# B&R Automation Studio project betaautomationstudio
Automation Studio 4.9.2.46; technology packages: Acp10Arnc0 5.12.2

## Configuration Config1

CPU X20CP1586, AutomationRuntime C4.90, Build 4.1.2, Vc V4.72.2

### Task classes (Cpu.sw)
```
Cyclic#4:
  control <- control.prg
  varUpdates <- varUpdates.prg
NcDataObjects: acp10etxen <- acp10etxen.dob, gAxisa <- gAxisobj.gAxisa.dob, gAxisi <- gAxisobj.gAxisi.dob
VcDataObjects: Visu <- Visu.dob
Libraries: Acp10man, Acp10par, NcGlobal, Acp10_MC, sys_lib, brsystem, runtime, Acp10sim
```

### Hardware
```
X20CP1586 : X20CP1586 v1.8.1.0
  Connector IF2:
    ActivateDevice = 1
    Vnc1
    VncVcObjectName1 = Visu
    VncKeyMappingFile1 = VC\PS2-Keyboard.dis
  ConfigurationID = betaprojectAS_Config1
  Simulation = 1
```

### Acp10cfg.ncc - X20CP1586/Motion/Acp10cfg.ncc
```
NcConfiguration (Version=5.12.2, NcSwId=Acp10)
  ACP10CF1_typ:
    cnt_nettrc_rec_drive = 1500
    bufsize_trace_upload = 1200
    tc_nc_man_task = Cyclic #1
    glob_pv_as_ncobject = Yes
    ncsys_dl_broadcast = Yes
    ncsys_dl_acp_reset = Yes
    safemc_log_err_to_ax = Yes
    network_init:
      ncsw_init_execute = Yes
      automatic_execute = No
      node_nr_warning = Yes
      net_err_before_ncact = Yes
    nettrc:
      enter_parsecrec = Yes
      enter_ncaction = Yes
      save_ring_startidx = Yes
    cam_prof_download:
      cam_dat_dl_parallel = No
      tc_cam_dl_parallel = Task class for NC Manager task
    plk_if[0]:
      if_name = IF3
      tc_CycDat_PLCopen = Task class for NC Manager task
      mc_broadcast_extdat = No
```

### Acp10map.ncm - X20CP1586/Motion/Acp10map.ncm
```
NcMapping (NcSwId=Acp10, DisabledNodesAreHidden=False)
  NcObject gAxis (ModuleId=8EIxxxMxS1x.xxxx-1, Type=ncAXIS, Channel=1, AcoposSimulation=Standard, InitParameter=gAxisi, AcoposParameter=gAxisa, Disabled=FALSE, ModuleDisabled=FALSE)
  NcObject 8EIxxxMxS1x.xxxx-1_ncV_AXIS1 (ModuleId=8EIxxxMxS1x.xxxx-1, Type=ncV_AXIS, Channel=1, Disabled=TRUE, ModuleDisabled=FALSE)
```

### PvMap.vvm - X20CP1586/PvMap.vvm
```iecst
VAR_CONFIG
	::pvi AT %Q.::pvi; (*PVI Variables, lol*)
END_VAR
```

## Logical view

Binary libraries used (declarations not repeated): operator, runtime, astime, AsIecCon, Acp10man 5.12.2, Acp10par 5.12.2, NcGlobal 5.12.2, Acp10_MC 5.12.2, sys_lib, brsystem, Acp10sim 5.12.2

### Global.typ - Global data types
```iecst
TYPE
	ctrlStateEnum :
		(
		CTRL_INIT,
		CTRL_OFF,
		CTRL_POWER_ON_AXIS,
		CTRL_POWERING_ON_AXIS,
		CTRL_POWER_OFF_AXIS,
		CTRL_POWERING_OFF_AXIS,
		CTRL_HOME_AXIS,
		CTRL_HOMING_AXIS,
		CTRL_STOPPING,
		CTRL_STANDSTILL,
		CTRL_MOVE_VELOCITY,
		CTRL_MOVE_ABSOLUTE,
		CTRL_ERROR,
		CTRL_MOVE_VELOCITY_ERROR,
		CTRL_MOVE_ABSOLUTE_ERROR,
		CTRL_FATAL_ERROR,
		CTRL_FATAL_ERROR_EXIT
	);

	mcBlocksType : STRUCT
		power : MC_Power;
		home : MC_Home;
		stop : MC_Stop;
		reset : MC_Reset;
		moveVelocity : MC_MoveVelocity;
		moveAbsolute : MC_MoveAbsolute;
		currentPosition : MC_ReadActualPosition;
		currentVelocity : MC_ReadActualVelocity;
		status : MC_ReadStatus;
		error : MC_ReadAxisError;
	END_STRUCT;

	gLocalPID : STRUCT
		enabled : BOOL;					(*  *)
		proportionalGain : BOOL;		(*  *)
		integralGain : BOOL;			(*  *)
		derivativeGain : BOOL;			(*  *)
	END_STRUCT;

	gControlType : STRUCT
		localPID : gLocalPID;			(*  *)
		modeVelocity : BOOL;			(*  *)
		setPosition : REAL;				(*  *)
		setDirection : BOOL;			(*  *)
		setVelocity : REAL;				(*  *)
		currentPosition : REAL;			(*  *)
		currentAngle : REAL;			(*  *)
		currentVelocity : REAL;			(*  *)
		currentDirection : INT;			(*  *)
		limitAcceleration : REAL := 1000;	(*  *)
		limitVelocity : REAL := 200;	(*  *)
		limitPosPos : DINT := -5000;	(*  *)
		limitNegPos : DINT := 5000;		(*  *)
	END_STRUCT;

	hmiType : STRUCT
		fields : vFieldType;			(*  *)
		indicators : vIndicatorType;	(*  *)
		buttons : vButtonType;			(*  *)
	END_STRUCT;

	vButtonType : STRUCT
		on : BOOL;						(*  *)
		onPrevious : BOOL;
		off : BOOL;						(*  *)
		offPrevious : BOOL;
		start : BOOL;					(*  *)
		startPrevious : BOOL;
		stop : BOOL;					(*  *)
		stopPrevious : BOOL;
		localPid : BOOL;				(*  *)
		localPidPrevious : BOOL;
		simulinkPid : BOOL;				(*  *)
		simulinkPidPrevious : BOOL;
		externalSim : BOOL;				(*  *)
		externalSimPrevious : BOOL;
		simulinkSim : BOOL;				(*  *)
		simulinkSimPrevious : BOOL;
		ackError : BOOL;				(*  *)
		ackErrorPrevious : BOOL;
		overridePosition : BOOL;		(*  *)
		overridePositionPrevious : BOOL;
	END_STRUCT;

	vFieldType : STRUCT
		velocity : REAL;			(*  *)
		position : REAL;			(*  *)
		angle : REAL;				(*  *)
		ovrPosition : REAL;			(*  *)
		accelerationLimit : REAL;	(*  *)
		velocityLimit : REAL;		(*  *)
		positionLimitNeg : DINT;	(*  *)
		positionLimitPos : DINT;	(*  *)
		controlState : WSTRING[40];	(*  *)
		errorCode : REAL;			(*  *)
		errorText : WSTRING[40];	(*  *)
	END_STRUCT;

	vIndicatorType : STRUCT
		power : INT;				(*  *)
		home : INT;					(*  *)
		stop : INT;					(*  *)
		reset : INT;				(*  *)
		moveVelocity : INT;			(*  *)
		movePosition : INT;			(*  *)
		readVelocity : INT;			(*  *)
		readPosition : INT;			(*  *)
		status : INT;				(*  *)
		error : INT;				(*  *)
		readParam : INT;			(*  *)
		writeParam : INT;			(*  *)
	END_STRUCT;

	opcuaWriteType : STRUCT 			(* For variables read from OPCUA *)
		cartPosition : REAL := 0.0;		(* mm *)
		cartVelocity : REAL := 0.0;		(* mm/s *)
		pendulumAngle : REAL := 0.0;	(* Rad, 0 is upright position *)
	END_STRUCT;
	opcuaReadType : STRUCT 				(* For variables written to OPCUA *)
		setCartVelocity : REAL := 0.0;	(* Negative is backward motion *)
	END_STRUCT;

	pviMotorType : STRUCT
		start : BOOL := FALSE;				(* Start the motor *)
		forward : BOOL := FALSE;			(* Set motor direction *)
		setVelocity : INT := 0;				(*  *)
		setConverterFrequency : INT := 0;	(*  *)
		isStarted : BOOL := FALSE;			(*  *)
		isStopped : BOOL := FALSE;			(*  *)
		isForward : BOOL := FALSE;			(*  *)
		isBackward : BOOL := FALSE;			(*  *)
		isMax : BOOL := FALSE;				(* Motor is at max limit *)
		isMiddle : BOOL := FALSE;			(* Motor is on exact middle *)
		isMin : BOOL := FALSE;				(* Motor is at min limit *)
		offsetMax : BOOL := FALSE;			(*  *)
		offsetMin : BOOL := FALSE;			(*  *)
		isReset : BOOL := FALSE;			(*  *)
		velocity : INT := 0;				(* Actual motor velocity *)
	END_STRUCT;

	pviType : STRUCT
		cartPositionEncoder : DINT := 0;	(* Cart position encoder output, currently in 1mm/units *)
		pendulumAngle : DINT := 0; 		(* Angle output, 1024 divisions per rotation *)
		motor : pviMotorType;		(* All motor specific variables *)
	END_STRUCT;

END_TYPE
```

### Global.var - Global variables
```iecst
VAR
	gAxis : ACP10AXIS_typ;			(* Required axis object *)

	ctrlState : ctrlStateEnum := CTRL_INIT;	(* Control loop state *)
	mc : mcBlocksType;				(* Function blocks for motor control *)

	gControl : gControlType;		(* Control related variables *)
	hmi : hmiType;					(* HMI stuff *)
	opcua_r : opcuaReadType;		(* Variables readable with OPCUA *)
	opcua_w : opcuaWriteType;		(* Variables writeable with OPCUA *)
	pvi : pviType;					(* Variables shared with PVI *)
END_VAR
```


### Data object Logical/acp10etxen (Ett)

- acp10etxen.ett (not shown)

### Package Logical/gAxisobj - gAxisobj

- Data object Logical/gAxisobj/gAxisa (Apt) (no source held here)

### Data object Logical/gAxisobj/gAxisi (Ax)

#### gAxisi.ax
```
InitParameter (Version=5.12.2, NcSwId=Acp10)
  ACP10AXIS_typ:
    dig_in:
      level:
        reference = ncACTIV_HI
        pos_hw_end = ncACTIV_HI
        neg_hw_end = ncACTIV_HI
        trigger1 = ncACTIV_HI
        trigger2 = ncACTIV_HI
    encoder_if:
      parameter:
        count_dir = ncSTANDARD
        scaling:
          load:
            units = 1000
            rev_motor = 1
    limit:
      parameter:
        v_pos = 10000
        v_neg = 10000
        a1_pos = 50000
        a2_pos = 50000
        a1_neg = 50000
        a2_neg = 50000
        t_jolt = 0
        t_in_pos = 0
        pos_sw_end = 2000000000
        neg_sw_end = -2000000000
        ds_warning = 500
        ds_stop = 1000
        a_stop = 1.0e30
        dv_stop = 0
        dv_stop_mode = ncOFF
    controller:
      mode = ncPOSITION
      position:
        kv = 50
        tn = 0
        t_predict = 0.0004
        t_total = 0.0004
        p_max = 1.0e30
        i_max = 0
      speed:
        kv = 2.0
        tn = 0
        t_filter = 0.0
        isq_filter1:
          type = ncOFF
          a0 = 0.0
          a1 = 0.0
          b0 = 0.0
          b1 = 0.0
          b2 = 0.0
          c0_par_id = 0
          c1_par_id = 0
        isq_filter2:
          type = ncOFF
          a0 = 0.0
          a1 = 0.0
          b0 = 0.0
          b1 = 0.0
          b2 = 0.0
          c0_par_id = 0
          c1_par_id = 0
        isq_filter3:
          type = ncOFF
          a0 = 0.0
          a1 = 0.0
          b0 = 0.0
          b1 = 0.0
          b2 = 0.0
          c0_par_id = 0
          c1_par_id = 0
      uf:
        type = ncLINEAR + ncCORRECTION
        auto_config = ncMOTOR_PAR
        u0 = 0
        un = 0
        fn = 50.0
        k_f_slip = 0
      ff:
        mode = ncSTANDARD
        torque_load = 0.0
        torque_pos = 0.0
        torque_neg = 0.0
        kv_torque = 0.0
        inertia = 0.0
        t_filter_a = 0.0
      fb:
        mode = ncSTANDARD
        speed_mix_ratio = 0.0
        speed_kv = 2.0
      model:
        mass1:
          inertia = 0
          viscous_friction = 0
        mass2:
          inertia = 0
          viscous_friction = 0
          stiffness = 0
          damping = 0
    move:
      stop:
        parameter[0]:
          decel_ramp = ncA_LIMIT
          controller = ncON
        parameter[1]:
          decel_ramp = ncA_LIMIT
          controller = ncON
        parameter[2]:
          decel_ramp = ncA_LIMIT
          controller = ncON
        parameter[3]:
          decel_ramp = ncA_LIMIT
          controller = ncON
        quickstop:
          decel_ramp = ncA_LIMIT
          t_jolt = 0
        drive_error:
          decel_ramp = ncA_LIMIT
      homing:
        parameter:
          s = 0
          v_switch = 5000
          v_trigger = 500
          a = 50000
          mode = ncDIRECT
          edge_sw = ncPOSITIVE
          start_dir = ncPOSITIVE
          trigg_dir = ncPOSITIVE
          ref_pulse = ncOFF
          fix_dir = ncOFF
          tr_s_block = 0
          torque_lim = 0
          ds_block = 0
          ds_stop = 0
      basis:
        parameter:
          v_pos = 5000
          v_neg = 5000
          a1_pos = 50000
          a2_pos = 50000
          a1_neg = 50000
          a2_neg = 50000
    message:
      text:
        parameter:
          format = ncBREAK
          columns = 80
          data_modul = acp10etxen
```

### Program Logical/control (IEC)

#### Variables.var
```iecst
VAR
	state : ctrlStateEnum := CTRL_INIT;
	mc : mcBlocksType;
END_VAR
```

#### Main.st
```iecst
PROGRAM _INIT
	(* Insert code here *)

END_PROGRAM

PROGRAM _CYCLIC
	CASE ctrlState OF
		CTRL_INIT:
			// Binding the motion axis to MC blocks
			mc.home.Axis := ADR(gAxis);
			mc.moveAbsolute.Axis := ADR(gAxis);
			mc.moveVelocity.Axis := ADR(gAxis);
			mc.power.Axis := ADR(gAxis);
			mc.reset.Axis := ADR(gAxis);
			mc.stop.Axis := ADR(gAxis);
			mc.currentPosition.Axis := ADR(gAxis);
			mc.currentVelocity.Axis := ADR(gAxis);
			mc.error.Axis := ADR(gAxis);

			// Next state
			ctrlState := CTRL_OFF;

		CTRL_OFF:
			// Check if ON is requested and change state
			IF hmi.buttons.on THEN
				ctrlState := CTRL_POWER_ON_AXIS;
			END_IF

		CTRL_POWER_ON_AXIS:
			// Enable the block required for std operation
			mc.power.Enable := TRUE;
			mc.currentPosition.Enable := TRUE;
			mc.currentVelocity.Enable := TRUE;
			mc.error.Enable := TRUE;
			mc.status.Enable := TRUE;

			// Change state
			ctrlState := CTRL_POWERING_ON_AXIS;

		CTRL_POWERING_ON_AXIS:
			// Change state if Power is on
			// TODO: Include checks for the other blocks?
			IF mc.power.Status THEN
				ctrlState := CTRL_HOME_AXIS;
			END_IF

		CTRL_POWER_OFF_AXIS:
			// Disable the blocks used for std operation
			mc.power.Enable := FALSE;
			mc.currentPosition.Enable := FALSE;
			mc.currentVelocity.Enable := FALSE;
			mc.error.Enable := FALSE;
			mc.status.Enable := FALSE;

			// Change state
			ctrlState := CTRL_POWERING_OFF_AXIS;

		CTRL_POWERING_OFF_AXIS:
			// Change state when block are off
			IF NOT mc.power.Status AND NOT mc.currentPosition.Valid AND NOT mc.currentVelocity.Valid THEN
				ctrlState := CTRL_OFF;
			END_IF

		CTRL_HOME_AXIS:
			// If Execute is true, flip and come back next cycle
			IF mc.home.Execute THEN
				mc.home.Execute := FALSE;
			ELSE
				// Start homing and change state
				mc.home.Execute := TRUE;
				ctrlState := CTRL_HOMING_AXIS;
			END_IF

		CTRL_HOMING_AXIS:
			// Change state when homing is done
			IF mc.home.Done THEN
				mc.home.Execute := FALSE;
				ctrlState := CTRL_STOPPING;
			END_IF

		CTRL_STOPPING:
			// Change state when confirmed stopped
			mc.stop.Execute := TRUE;
			IF mc.stop.Done THEN
				mc.stop.Execute := FALSE;
				ctrlState := CTRL_STANDSTILL;
			END_IF

		CTRL_STANDSTILL:
			// Wait for something to start the operation
			IF hmi.buttons.start OR hmi.buttons.overridePosition THEN
				// Reset the button
				hmi.buttons.start := FALSE;
				// If the override move position is active, do that
				IF hmi.buttons.overridePosition THEN
					// Set the move position from the field
					gControl.setPosition := hmi.fields.ovrPosition;
					// Reset the button
					hmi.buttons.overridePosition := FALSE;
					// Change to move absolute state
					ctrlState := CTRL_MOVE_ABSOLUTE;
				ELSE
					// 'Normal' velocity based operation
					ctrlState := CTRL_MOVE_VELOCITY;
				END_IF
			ELSIF hmi.buttons.off THEN
				// Power off if button has been pushed
				hmi.buttons.off := FALSE;
				ctrlState := CTRL_POWER_OFF_AXIS;
			END_IF

		CTRL_MOVE_VELOCITY:
			// Check if a stop or manual position override is requested
			IF hmi.buttons.stop OR hmi.buttons.overridePosition THEN
				// Reset button
				hmi.buttons.stop := FALSE;
				// Stop velocity block and change to stop state
				mc.moveVelocity.Execute := FALSE;
				ctrlState := CTRL_STOPPING;
			ELSE
				// Check that velocity requested is within limits
				IF gControl.setVelocity >= 0 AND gControl.setVelocity < gControl.limitVelocity THEN
					// Update move block velocity
					mc.moveVelocity.Velocity := gControl.setVelocity;
					// Set direction
					IF gControl.setDirection THEN
						mc.moveVelocity.Direction := mcPOSITIVE_DIR;
					ELSE
						mc.moveVelocity.Direction := mcNEGATIVE_DIR;
					END_IF

					// Toggle execute and update the block to allow for changes in same cycle
					IF mc.moveVelocity.Execute THEN
						mc.moveVelocity.Execute := FALSE;
						mc.moveVelocity();
					END_IF
					// Start executing move
					mc.moveVelocity.Execute := TRUE;
				ELSE
					// Limits not met, stop motion
					mc.moveVelocity.Velocity := 0;
					mc.moveVelocity.Execute := FALSE;
					ctrlState := CTRL_STOPPING;
				END_IF
			END_IF

		CTRL_MOVE_ABSOLUTE:
			// This move mode is used for the override position only
			IF hmi.buttons.stop THEN
				// Reset the button
				hmi.buttons.stop := FALSE;
				// Stop moving
				mc.moveAbsolute.Execute := FALSE;
				ctrlState := CTRL_STOPPING;
			ELSIF mc.moveAbsolute.Done THEN
				// Movement complete, go to standstill state
				mc.moveAbsolute.Execute := FALSE;
				ctrlState := CTRL_STANDSTILL;
			ELSE
				// Check if move is needed (within 0.1 unit of current position)
				IF ABS(gControl.currentPosition - gControl.setPosition) > 0.1 THEN
					// Set new position in block
					mc.moveAbsolute.Position := gControl.setPosition;
					// Start execution
					mc.moveAbsolute.Execute := TRUE;
				ELSIF NOT mc.moveAbsolute.Execute THEN
					// Move not big enough, go to standstill state
					// If block is already active we might just be very close and don't want to do anything
					mc.moveAbsolute.Execute := FALSE;
					ctrlState := CTRL_STANDSTILL;
				END_IF
			END_IF

		CTRL_ERROR:

		CTRL_FATAL_ERROR:

		CTRL_FATAL_ERROR_EXIT:

	END_CASE

	// Updating blocks, minus info-only blocks (see varUpdates loop)
	mc.home();
	mc.moveAbsolute();
	mc.moveVelocity();
	mc.power();
	mc.reset();
	mc.stop();

	// Error checking
	// TODO: Do something
	IF mc.home.Error THEN
	END_IF
	IF mc.moveAbsolute.Error THEN
	END_IF
	IF mc.moveVelocity.Error THEN
	END_IF
	IF mc.power.Error THEN
	END_IF
	IF mc.reset.Error THEN
	END_IF
	IF mc.stop.Error THEN
	END_IF
	IF mc.currentPosition.Error THEN
	END_IF
	IF mc.currentVelocity.Error THEN
	END_IF
	IF mc.status.Error THEN
	END_IF

END_PROGRAM

PROGRAM _EXIT
	(* Insert code here *)

END_PROGRAM
```

- Visualisation Logical/Visu (not shown)

### Program Logical/varUpdates (IEC)

#### Main.st
```iecst
PROGRAM _INIT
	(* Insert code here *)

END_PROGRAM

PROGRAM _CYCLIC
	// Clearing errorText if ack'ed
	IF hmi.buttons.ackError THEN
		// Reset button
		hmi.buttons.ackError := FALSE;
		// Acknowledge error
		mc.error.Acknowledge := TRUE;
	END_IF

	// Update the function blocks used for errors and reading values
	mc.currentPosition();
	mc.currentVelocity();
	mc.status();
	mc.error();

	// Some HMI button logic for determining which sim and PID to use
	IF hmi.buttons.externalSim AND NOT hmi.buttons.externalSimPrevious THEN
		// Mode switched to external sim
		hmi.buttons.externalSimPrevious := hmi.buttons.externalSim;
		hmi.buttons.simulinkSim := NOT hmi.buttons.externalSim;
		hmi.buttons.simulinkSimPrevious := NOT hmi.buttons.externalSim;
	END_IF
	IF hmi.buttons.simulinkSim AND NOT hmi.buttons.simulinkSimPrevious THEN
		// Mode switched to simulink sim
		hmi.buttons.simulinkSimPrevious := hmi.buttons.simulinkSim;
		hmi.buttons.externalSim := NOT hmi.buttons.simulinkSim;
		hmi.buttons.externalSimPrevious := NOT hmi.buttons.simulinkSim;
	END_IF

	IF hmi.buttons.localPid AND NOT hmi.buttons.localPidPrevious THEN
		// Mode switched to local PID
		hmi.buttons.localPidPrevious := hmi.buttons.localPid;
		hmi.buttons.simulinkPid := NOT hmi.buttons.localPid;
		hmi.buttons.simulinkPidPrevious := NOT hmi.buttons.localPid;
	END_IF
	IF hmi.buttons.simulinkPid AND NOT hmi.buttons.simulinkPidPrevious THEN
		// Mode switched to simulink PID
		hmi.buttons.simulinkPidPrevious := hmi.buttons.simulinkPid;
		hmi.buttons.localPid := NOT hmi.buttons.simulinkPid;
		hmi.buttons.localPidPrevious := NOT hmi.buttons.simulinkPid;
	END_IF

	// Update variables from motor position, velocity, and pendulum angle
	gControl.currentAngle := 0; // TODO: Where do I get this?
	gControl.currentPosition := mc.currentPosition.Position;
	gControl.currentVelocity := mc.currentVelocity.Velocity;
	gControl.currentDirection := mc.moveVelocity.Direction;

	// Update variables from simulation through PVI
	IF hmi.buttons.externalSim THEN
		// Read the current pendulum angle and cart position? from PVI
		// TODO: Scale this correctly
		gControl.currentAngle := DINT_TO_REAL(pvi.pendulumAngle);
		// TODO: I don't think we should let pvi override the MC block position?
		//gControl.currentPosition := pvi.cartPositionEncoder;
		// Write the current motor state, direction and velocity to PVI
		pvi.motor.start := mc.moveVelocity.Execute;
		pvi.motor.setVelocity := REAL_TO_INT(mc.moveVelocity.Velocity);
		IF mc.moveVelocity.Direction = mcPOSITIVE_DIR THEN
			pvi.motor.forward := TRUE;
		ELSE
			pvi.motor.forward := FALSE;
		END_IF

	END_IF
	// Update variables for simulink simulation
	IF hmi.buttons.simulinkSim THEN
		// Read the current pendulum angle from OPCUA
		gControl.currentAngle := opcua_w.pendulumAngle;
		// Write the position and cart velocity to OPCUA
		// TODO: Scale the written velocity correctly
		opcua_w.cartPosition := gControl.currentPosition;
		opcua_w.cartVelocity := gControl.currentVelocity;
	END_IF

	// Update variables for local PID control?
	IF hmi.buttons.localPid THEN
	END_IF
	// Update variables for simulink PID control
	IF hmi.buttons.simulinkPid THEN
		// Write the current position and angle
		// Read the new setVelocity
		gControl.setVelocity := opcua_r.setCartVelocity;
		// Write the current position and pendulum angle to OPCUA
		opcua_w.cartPosition := gControl.currentPosition;
		// TODO: Map the velocity correctly
		opcua_w.cartVelocity := gControl.currentVelocity;
		opcua_w.pendulumAngle := gControl.currentAngle;
	END_IF

	// Set movement limits from gControl struct
	mc.moveAbsolute.Acceleration := gControl.limitAcceleration;
	mc.moveAbsolute.Deceleration := gControl.limitAcceleration;
	mc.moveAbsolute.Velocity := gControl.limitVelocity;
	mc.moveVelocity.Acceleration := gControl.limitAcceleration;
	mc.moveVelocity.Deceleration := gControl.limitAcceleration;

	// And an error block thing
	mc.error.Acknowledge := FALSE;

	// Update HMI fields and indicators
	CASE ctrlState OF
		CTRL_INIT:
			hmi.fields.controlState := "CTRL_INIT";
		CTRL_OFF:
			hmi.fields.controlState := "CTRL_OFF";
		CTRL_POWER_ON_AXIS:
			hmi.fields.controlState := "CTRL_POWER_ON_AXIS";
		CTRL_POWERING_ON_AXIS:
			hmi.fields.controlState := "CTRL_POWERING_ON_AXIS";
		CTRL_POWER_OFF_AXIS:
			hmi.fields.controlState := "CTRL_POWER_OFF_AXIS";
		CTRL_POWERING_OFF_AXIS:
			hmi.fields.controlState := "CTRL_POWERING_OFF_AXIS";
		CTRL_HOME_AXIS:
			hmi.fields.controlState := "CTRL_HOME_AXIS";
		CTRL_HOMING_AXIS:
			hmi.fields.controlState := "CTRL_HOMING_AXIS";
		CTRL_STOPPING:
			hmi.fields.controlState := "CTRL_STOPPING";
		CTRL_STANDSTILL:
			hmi.fields.controlState := "CTRL_STANDSTILL";
		CTRL_MOVE_VELOCITY:
			hmi.fields.controlState := "CTRL_MOVE_VELOCITY";
		CTRL_MOVE_ABSOLUTE:
			hmi.fields.controlState := "CTRL_MOVE_ABSOLUTE";
		CTRL_ERROR:
			hmi.fields.controlState := "CTRL_ERROR";
		CTRL_FATAL_ERROR:
			hmi.fields.controlState := "CTRL_FATAL_ERROR";
		CTRL_FATAL_ERROR_EXIT:
			hmi.fields.controlState := "CTRL_FATAL_ERROR_EXIT";
		ELSE
			hmi.fields.controlState := "State fell through HMI Case!";
	END_CASE

	hmi.fields.errorCode := mc.error.ErrorID;
	hmi.fields.errorText := STRING_TO_WSTRING(mc.error.DataObjectName);

	hmi.fields.accelerationLimit := gControl.limitAcceleration;
	hmi.fields.velocityLimit := gControl.limitVelocity;
	hmi.fields.positionLimitPos := gControl.limitNegPos;
	hmi.fields.positionLimitNeg := gControl.limitPosPos;

	hmi.fields.angle := gControl.currentAngle;
	hmi.fields.position := gControl.currentPosition;
	hmi.fields.velocity := gControl.currentVelocity;

	hmi.indicators.power := mc.power.Error OR NOT mc.power.Enable;
	hmi.indicators.home := mc.home.Error OR NOT mc.home.Busy;
	hmi.indicators.stop := mc.stop.Error OR NOT mc.stop.Busy;
	hmi.indicators.reset := mc.reset.Error OR NOT mc.reset.Execute;
	hmi.indicators.moveVelocity := mc.moveVelocity.Error OR NOT mc.moveVelocity.Execute;
	hmi.indicators.movePosition := mc.moveAbsolute.Error OR NOT mc.moveAbsolute.Execute;
	hmi.indicators.readVelocity := mc.currentVelocity.Error OR NOT mc.currentVelocity.Enable;
	hmi.indicators.readPosition := mc.currentPosition.Error OR NOT mc.currentPosition.Enable;
	hmi.indicators.status := mc.status.Error AND NOT mc.status.Enable;
	hmi.indicators.error := mc.error.Error AND NOT mc.error.Enable;

END_PROGRAM

PROGRAM _EXIT
	(* Insert code here *)

END_PROGRAM
```

### Program Logical/Program

#### Types.typ
```iecst
TYPE
	controlStateEnum : (
		CTRL_INIT,
		CTRL_HOME_START,
		CTRL_HOME_SEEK_NEG,
		CTRL_HOME_SEEK_POS,
		CTRL_HOME_CENTER,
		CTRL_STOP,
		CTRL_RUNNING,
		CTRL_NO_SIM,
		CTRL_NO_CONTROLLER
	);

	opcuaType : STRUCT 			(* For OPCUA *)
		cartPosition : REAL := 0.0;		(* mm *)
		cartVelocity : REAL := 0.0;		(* mm/s *)
		pendulumAngle : REAL := 0.0;	(* Rad, 0 is upright position *)
		setCartVelocity : REAL := 0.0;	(* Negative is backward motion *)
	END_STRUCT;

	pviMotorType : STRUCT
		start : BOOL := FALSE;				(* Start the motor *)
		forward : BOOL := FALSE;			(* Set motor direction *)
		setVelocity : INT := 0;				(*  *)
		setConverterFrequency : INT := 0;	(*  *)
		isStarted : BOOL := FALSE;			(*  *)
		isStopped : BOOL := FALSE;			(*  *)
		isForward : BOOL := FALSE;			(*  *)
		isBackward : BOOL := FALSE;			(*  *)
		isMax : BOOL := FALSE;				(* Motor is at max limit *)
		isMiddle : BOOL := FALSE;			(* Motor is on exact middle *)
		isMin : BOOL := FALSE;				(* Motor is at min limit *)
		offsetMax : BOOL := FALSE;			(*  *)
		offsetMin : BOOL := FALSE;			(*  *)
		isReset : BOOL := FALSE;			(*  *)
		velocity : INT := 0;				(* Actual motor velocity *)
	END_STRUCT;

	pviType : STRUCT
		cartPositionEncoder : DINT := 0;	(* Cart position encoder output, currently in 1mm/units *)
		pendulumAngle : DINT := 0; 		(* Angle output, 1024 divisions per rotation *)
		motor : pviMotorType;			(* All motor specific variables *)
	END_STRUCT;

	controlType : STRUCT
		state : controlStateEnum;		(*  *)
		setVelocity : REAL;				(*  *)
		setPosition : REAL := 0;
		setPointPosition : REAL := 0;
		setAngle : REAL := 0;
		currentPosition : REAL;			(*  *)
		currentAngle : REAL;			(*  *)
		currentVelocity : REAL;			(*  *)
		currentAngularVelocity : REAL;
		currentDirection : BOOL;		(*  *)
		limitAcceleration : REAL := 1000;	(*  *)
		limitVelocity : REAL := 20000;	(*  *)
		limitPosPos : DINT := -5000;	(*  *)
		limitNegPos : DINT := 5000;		(*  *)
		homing : homingType;		(*  *)
	END_STRUCT;

	localLqrType : STRUCT
		A : ARRAY[1..4, 1..4] OF LREAL :=
		0, 1, 0, 0,
		0, -10, 1.6498, -0.0134,
		0, 0, 0, 1,
		0, -55.8140, 64.0173, -0.5198;
		B : ARRAY[1..4] OF LREAL := 0, 2, 0, 11.1628;
		Kf : ARRAY[1..4, 1..2] OF LREAL :=
		-3.1768, -0.0803,
		-0.0491, -1.2372,
		-0.0803, -15.3344,
		-0.2485, -112.5752;
		Klqr2 : ARRAY[1..4] OF LREAL := -3.3541, -12.8984, 57.1684, 16.7280;

		Klqr : ARRAY[1..4] OF LREAL := 2.5683, 9.3490, -38.5829, -12.4979;

		u : LREAL := 0;

		x : ARRAY[1..4] OF LREAL := 0,0,0,0;
		xn : ARRAY[1..4] OF LREAL := 0,0,0,0;

		intOut : ARRAY[1..4] OF LREAL := 0,0,0,0;
		intSave : ARRAY[1..4] OF LREAL := 0,0,0,0;

		mc : LREAL := 0.5;
		mp : LREAL := 0.084;
		Ts : LREAL := 0.01;
	END_STRUCT;

	homingType : STRUCT
		foundNegLim : REAL;				(*  *)
		foundPosLim : REAL;				(*  *)
		seekVelocity : REAL := 500;		(*  *)
		middleVelocity : REAL := 1500;	(*  *)
	END_STRUCT;

	hmiType : STRUCT
		fields : hmiFieldType;			(*  *)
		indicators : hmiIndicatorType;	(*  *)
		buttons : hmiButtonType;			(*  *)

	END_STRUCT;

	hmiButtonType : STRUCT
		start : BOOL;					(*  *)
		startPrevious : BOOL;
		localPid : BOOL;				(*  *)
		localPidPrevious : BOOL;
		simulinkPid : BOOL;				(*  *)
		simulinkPidPrevious : BOOL;
		experiorSim : BOOL;				(*  *)
		experiorSimPrevious : BOOL;
		simulinkSim : BOOL;				(*  *)
		simulinkSimPrevious : BOOL;
	END_STRUCT;

	hmiFieldType : STRUCT
		velocity : REAL;			(*  *)
		position : REAL;			(*  *)
		angle : REAL;				(*  *)
		ovrPosition : REAL;			(*  *)
		accelerationLimit : REAL;		(*  *)
		velocityLimit : REAL;			(*  *)
		positionLimitNeg : REAL;		(*  *)
		positionLimitPos : REAL;		(*  *)
		controlState : WSTRING[40];		(*  *)
	END_STRUCT;

	hmiIndicatorType : STRUCT
		pvi : BOOL; 	(*  *)
		opcua : BOOL;	(*  *)
	END_STRUCT;

END_TYPE
```

#### Variables.var
```iecst
VAR
	control : controlType;
	hmi : hmiType;
	opcua : opcuaType;
	pvi : pviType;
	lqr : localLqrType;
END_VAR
```

#### Main.st
```iecst
PROGRAM _INIT

	// Start in local mode with experior sim
	hmi.buttons.start := TRUE;
	hmi.buttons.experiorSim := TRUE;
	hmi.buttons.localPid := TRUE;

END_PROGRAM

PROGRAM _CYCLIC
	// 1. BUTTON LOGIC
	// 2. SIMULATION READS
	// 3. STATE SWITCH
	// 	3.1 HOMING
	//	3.2 SEEK TO MID
	//	3.3 CONTROL LOOP MODE
	// 4. SIMULATION WRITES
	// 5. HMI

	//////////////////
	// BUTTON LOGIC //
	//////////////////
	// Experior simulation button
	IF hmi.buttons.experiorSim AND NOT hmi.buttons.experiorSimPrevious THEN
		// Mode switched to experior sim
		hmi.buttons.experiorSimPrevious := hmi.buttons.experiorSim;
		hmi.buttons.simulinkSim := NOT hmi.buttons.experiorSim;
		hmi.buttons.simulinkSimPrevious := NOT hmi.buttons.experiorSim;
	ELSIF NOT hmi.buttons.experiorSim AND hmi.buttons.experiorSimPrevious THEN
		// Switched off
		hmi.buttons.experiorSimPrevious := hmi.buttons.experiorSim;
	END_IF

	// Simulink simulation button
	IF hmi.buttons.simulinkSim AND NOT hmi.buttons.simulinkSimPrevious THEN
		// Mode switched to simulink sim
		hmi.buttons.simulinkSimPrevious := hmi.buttons.simulinkSim;
		hmi.buttons.experiorSim := NOT hmi.buttons.simulinkSim;
		hmi.buttons.experiorSimPrevious := NOT hmi.buttons.simulinkSim;
	ELSIF NOT hmi.buttons.simulinkSim AND hmi.buttons.simulinkSimPrevious THEN
		// Switched off
		hmi.buttons.simulinkSimPrevious := hmi.buttons.simulinkSim;
	END_IF

	// Local control button
	IF hmi.buttons.localPid AND NOT hmi.buttons.localPidPrevious THEN
		// Mode switched to local PID
		hmi.buttons.localPidPrevious := hmi.buttons.localPid;
		hmi.buttons.simulinkPid := NOT hmi.buttons.localPid;
		hmi.buttons.simulinkPidPrevious := NOT hmi.buttons.localPid;
	ELSIF NOT hmi.buttons.localPid AND hmi.buttons.localPidPrevious THEN
		// Switched off
		hmi.buttons.localPidPrevious := hmi.buttons.localPid;
	END_IF

	// Simulink control button
	IF hmi.buttons.simulinkPid AND NOT hmi.buttons.simulinkPidPrevious THEN
		// Mode switched to simulink PID
		hmi.buttons.simulinkPidPrevious := hmi.buttons.simulinkPid;
		hmi.buttons.localPid := NOT hmi.buttons.simulinkPid;
		hmi.buttons.localPidPrevious := NOT hmi.buttons.simulinkPid;
	ELSIF NOT hmi.buttons.simulinkPid AND hmi.buttons.simulinkPidPrevious THEN
		// Switched off
		hmi.buttons.simulinkPidPrevious := hmi.buttons.simulinkPid;
	END_IF

	// Button logic for start button
	IF hmi.buttons.start AND NOT hmi.buttons.startPrevious THEN
		// Mode switched to ON
		hmi.buttons.startPrevious := hmi.buttons.start;
	ELSIF NOT hmi.buttons.start AND hmi.buttons.startPrevious THEN
		// Switched off
		hmi.buttons.startPrevious := hmi.buttons.start;
	END_IF
	//////////////////////
	// BUTTON LOGIC END //
	//////////////////////

	//////////////////////
	// SIMULATION READS //
	//////////////////////
	// Update the current values through either pvi or opcua, based on button states
	IF hmi.buttons.experiorSim THEN

		control.currentAngle := DINT_TO_REAL(pvi.pendulumAngle);
		control.currentPosition := DINT_TO_REAL(pvi.cartPositionEncoder) / 1000;
		// Remap angle so that 0 is vertical and signed, in radians
		control.currentAngle := (DINT_TO_REAL(pvi.pendulumAngle)) * 2 * 3.14159 / 1024.0;
		IF control.currentAngle > 3.14159 THEN
			control.currentAngle := control.currentAngle - 2 * 3.14159;
		END_IF
		// Flip it
		control.currentAngle := -control.currentAngle;

		// And direction, velocity is just signed
		IF control.currentVelocity >= 0 THEN
			control.currentDirection := TRUE;
		ELSE
			control.currentDirection := FALSE;
		END_IF

	ELSIF hmi.buttons.simulinkSim THEN
		// Same stuff, but for simulink
		control.currentAngle := opcua.pendulumAngle;
		control.currentPosition := opcua.cartPosition;
		control.currentVelocity := opcua.cartVelocity;
		IF control.currentVelocity >= 0 THEN
			control.currentDirection := TRUE;
		ELSE
			control.currentDirection := FALSE;
		END_IF

	ELSE
		// No simulation is chosen, zero out
		control.currentAngle := 0;
		control.currentPosition := 0;
		control.currentVelocity := 0;
		control.currentDirection := FALSE;

	END_IF
	/////////////////////////
	// SIMULATION READ END //
	/////////////////////////

	//////////////////
	// STATE SWITCH //
	//////////////////
	CASE control.state OF
		CTRL_INIT:
			// Hmm ...
			//control.state := CTRL_HOME_START;
			control.state := CTRL_RUNNING;

			lqr.x[1] := 0;
			lqr.x[2] := 0;
			lqr.x[3] := 0;
			lqr.x[4] := 0;
			lqr.xn := lqr.x;
			lqr.intOut := lqr.x;
			lqr.intSave := lqr.x;
			lqr.u := 0;

		CTRL_HOME_START:
			// There's only homing for Experior
			// Matlab gets a set of default values
			IF hmi.buttons.experiorSim THEN
				control.state := CTRL_HOME_SEEK_NEG;
			ELSIF hmi.buttons.simulinkSim THEN
				control.state := CTRL_STOP;
			END_IF

		CTRL_HOME_SEEK_NEG:
			// Seek the negative limit switch
			IF hmi.buttons.experiorSim THEN
				control.setVelocity := -control.homing.seekVelocity;
				IF pvi.motor.isMin THEN
					control.homing.foundNegLim := control.currentPosition;
					control.state := CTRL_HOME_SEEK_POS;
				END_IF

			ELSIF hmi.buttons.simulinkSim THEN
				// TODO: Implement some homing for simulink
				control.state := CTRL_STOP;

			ELSE
				// No sim, wat do
				control.state := CTRL_NO_SIM;

			END_IF;

		CTRL_HOME_SEEK_POS:
			// Seek the positive limit switch
			IF hmi.buttons.experiorSim THEN
				control.setVelocity := control.homing.seekVelocity;
				IF pvi.motor.isMax THEN
					control.homing.foundPosLim := control.currentPosition;
					control.state := CTRL_HOME_CENTER;
				END_IF

			ELSIF hmi.buttons.simulinkSim THEN
				// TODO: Implement some homing for simulink
				control.state := CTRL_STOP;

			ELSE
				// No sim, wat do
				control.state := CTRL_NO_SIM;

			END_IF;

		CTRL_HOME_CENTER:
			// Move to the center position to prep for start
			IF hmi.buttons.experiorSim THEN
				control.setVelocity := -control.homing.middleVelocity;
				IF pvi.motor.isMiddle OR ((control.homing.foundNegLim + control.homing.foundPosLim)/2 >= control.currentPosition) THEN
					control.state := CTRL_STOP;
				END_IF

			ELSIF hmi.buttons.simulinkSim THEN
				// TODO: Implement some homing for simulink
				control.state := CTRL_STOP;

			ELSE
				// No sim, wat do
				control.state := CTRL_NO_SIM;

			END_IF;

		CTRL_STOP:
			// Wait here until started
			control.setVelocity := 0;
			IF hmi.buttons.start THEN
				control.state := CTRL_RUNNING;
			END_IF

		CTRL_RUNNING:
			// Check if no longer started
			IF NOT hmi.buttons.start THEN
				control.state := CTRL_STOP;

			ELSE
				//////////////////
				// CONTROL LOOP //
				//////////////////
				IF hmi.buttons.localPid THEN
					// This is where the local control can be calculated
					// The calculated velocity is set through control.setVelocity

					//lqr.x[1] := lqr.x[1] - control.setPosition;
					//lqr.x[2];
					//lqr.x[3] := lqr.x[3] - control.setAngle;
					//lqr.x[4]];

					lqr.u := lqr.Klqr[1] * (lqr.x[1] - control.setPosition) + lqr.Klqr[2] * lqr.x[2] + lqr.Klqr[3] * (lqr.x[3] - control.setAngle) + lqr.Klqr[4] * lqr.x[4];

					control.setVelocity := LREAL_TO_REAL(lqr.u * (1 / (lqr.mc + lqr.mp)) * lqr.Ts) * 1000;

					lqr.xn[1] := lqr.B[1] * lqr.u + lqr.A[1,1] * lqr.x[1] + lqr.A[1,2] * lqr.x[2] + lqr.A[1,3] * lqr.x[3] + lqr.A[1,4] * lqr.x[4] + lqr.Kf[1,2] * (lqr.x[3] - control.currentAngle) + lqr.Kf[1,1] * (lqr.x[1] - control.currentPosition);
					lqr.xn[2] := lqr.B[2] * lqr.u + lqr.A[2,1] * lqr.x[1] + lqr.A[2,2] * lqr.x[2] + lqr.A[2,3] * lqr.x[3] + lqr.A[2,4] * lqr.x[4] + lqr.Kf[2,2] * (lqr.x[3] - control.currentAngle) + lqr.Kf[2,1] * (lqr.x[1] - control.currentPosition);
					lqr.xn[3] := lqr.B[3] * lqr.u + lqr.A[3,1] * lqr.x[1] + lqr.A[3,2] * lqr.x[2] + lqr.A[3,3] * lqr.x[3] + lqr.A[3,4] * lqr.x[4] + lqr.Kf[3,2] * (lqr.x[3] - control.currentAngle) + lqr.Kf[3,1] * (lqr.x[1] - control.currentPosition);
					lqr.xn[4] := lqr.B[4] * lqr.u + lqr.A[4,1] * lqr.x[1] + lqr.A[4,2] * lqr.x[2] + lqr.A[4,3] * lqr.x[3] + lqr.A[4,4] * lqr.x[4] + lqr.Kf[4,2] * (lqr.x[3] - control.currentAngle) + lqr.Kf[4,1] * (lqr.x[1] - control.currentPosition);

					lqr.intOut[1] := (lqr.xn[1] * lqr.Ts/2) + lqr.intSave[1];
					lqr.intOut[2] := (lqr.xn[2] * lqr.Ts/2) + lqr.intSave[2];
					lqr.intOut[3] := (lqr.xn[3] * lqr.Ts/2) + lqr.intSave[3];
					lqr.intOut[4] := (lqr.xn[4] * lqr.Ts/2) + lqr.intSave[4];

					lqr.intSave[1] := lqr.intOut[1] + (lqr.xn[1] * lqr.Ts / 2);
					lqr.intSave[2] := lqr.intOut[2] + (lqr.xn[2] * lqr.Ts / 2);
					lqr.intSave[3] := lqr.intOut[3] + (lqr.xn[3] * lqr.Ts / 2);
					lqr.intSave[4] := lqr.intOut[4] + (lqr.xn[4] * lqr.Ts / 2);

					lqr.x[1] := lqr.intOut[1];
					lqr.x[2] := lqr.intOut[2];
					lqr.x[3] := lqr.intOut[3];
					lqr.x[4] := lqr.intOut[4];

				ELSIF hmi.buttons.simulinkPid THEN
					// Simulink has the calculated value for velocity
					control.setVelocity := opcua.setCartVelocity;

					// Update the opcua from current simulated reads
					opcua.cartPosition := control.currentPosition;
					opcua.cartVelocity := control.currentVelocity;
					opcua.pendulumAngle := control.currentAngle;
				ELSE
					// No control is set
					control.setVelocity := 0;

				END_IF
				//////////////////////
				// CONTROL LOOP END //
				//////////////////////

			END_IF

		CTRL_NO_SIM:

		CTRL_NO_CONTROLLER:

	END_CASE;
	//////////////////////
	// STATE SWITCH END //
	//////////////////////

	///////////////////////
	// SIMULATION WRITES //
	///////////////////////
	IF hmi.buttons.experiorSim THEN
		// Force the motor controls active
		pvi.motor.start := TRUE;
		pvi.motor.forward := control.currentDirection;

		// Set the motor velocity from the control type
		IF control.setVelocity > 0 AND control.setVelocity > control.limitVelocity THEN
			pvi.motor.setVelocity := REAL_TO_INT(control.limitVelocity);
		ELSIF control.setVelocity < 0 AND -control.setVelocity > control.limitVelocity THEN
			pvi.motor.setVelocity := -REAL_TO_INT(control.limitVelocity);
		ELSE
			pvi.motor.setVelocity := REAL_TO_INT(control.setVelocity);
		END_IF

	ELSIF hmi.buttons.simulinkSim THEN
		// Write the calculated velocity to the opcua type
		opcua.setCartVelocity := control.setVelocity;

	END_IF
	//////////////////////////
	// SIMULATION WRITE END //
	//////////////////////////

	//////////////////
	// HMI UPDATING //
	//////////////////
	hmi.fields.angle := control.currentAngle;
	hmi.fields.position := control.currentPosition;
	hmi.fields.velocity := control.currentVelocity;
	hmi.fields.positionLimitPos := control.homing.foundPosLim;
	hmi.fields.positionLimitNeg := control.homing.foundNegLim;
	hmi.fields.controlState := "Hello!";

	//////////////////////
	// HMI UPDATING END //
	//////////////////////

END_PROGRAM

PROGRAM _EXIT
	(* Insert code here *)

END_PROGRAM
```
